TYPE ST_Signal_HMI :
STRUCT
	aIL	 : ARRAY[1..3] OF ARRAY[1..cOversamples*cScaleHMI] OF LREAL;
	aUL	 : ARRAY[1..3] OF ARRAY[1..cOversamples*cScaleHMI] OF LREAL;
END_STRUCT
END_TYPE

(* stored: Version 1.1.0.1, ProductVersion 3.1.4024.12
   DUT ST_Signal_HMI: Id {47927bc7-d342-450a-8839-bc5d8a72f9e3} *)
